FUNCTION_BLOCK FB_Teacher
VAR
    _sName : STRING := '';  
	sOutput : STRING := '';
END_VAR

PROPERTY Name : STRING
GET
//GET
Name := _sName;
END_GET
SET
// SET
_sName := Name;
END_SET
END_PROPERTY

METHOD teach
VAR_INPUT
	 pStudent : POINTER TO FB_Student;
END_VAR
sOutput := CONCAT(CONCAT(_sName, ' teaches '), pStudent^.Name);
END_METHOD

END_FUNCTION_BLOCK

(* stored: Version 1.1.0.1, ProductVersion 3.1.4024.16
   POU FB_Teacher: Id {16c507c1-b16e-46ba-bf73-a161bb7277e7}, SpecialFunc None
   Property Name: Id {6911d694-525c-4584-b3f8-46c3cdd6e170}
   Get Get: Id {37c7479e-95c6-4bc5-a301-3e61a0e06d38}
   Set Set: Id {2952892b-5c02-45da-902b-4a5f5a21f212}
   Method teach: Id {2c8dd030-0271-4730-b327-9550617c7756} *)
